TYPE ST_CapacitorSchemaColorBase :
STRUCT
	TopLineColor : E_LineColors;
	BottomLineColor : E_LineColors;
	BottomLineColor2 : E_LineColors;
	CapacitorColor : E_LineColors;
	GroundColor : E_LineColors;
END_STRUCT
END_TYPE

(* stored: Version 1.1.0.1, ProductVersion 3.1.4024.13
   DUT ST_CapacitorSchemaColorBase: Id {e00471a5-3e37-4e81-96a2-985bfb86df37} *)
